PROGRAM MAIN
VAR
END_VAR

END_PROGRAM

(* stored: Version 1.1.0.1
   POU MAIN: Id {1d6ded7b-eec9-4d4f-90a4-0e184fc63e5a} *)
